INTERFACE ITcoObjectRestorer

(*~
	<docu>
		<summary>
			Ensures calling the <c>Restore()</c> method on the object entered.
			<para>
				<example>
				<note type="Example">
				<para>
					Possibility to use the fluent syntax.
				</para>
					<code>ChangeState(newState).RestoreObject(myFirstChildObject).RestoreObject(mySecondChildObject);</code>
				 </note>
				</example>
			</para>
		</summary>
	</docu>
~*)
METHOD RestoreObject : ITcoObjectRestorer
VAR_INPUT
	Obj : ITcoRestorable;
END_VAR
END_METHOD

END_INTERFACE

(* stored: Version 1.1.0.1
   Itf ITcoObjectRestorer: Id {0b3638df-96b7-05c9-2091-ef8947995aad}
   Method RestoreObject: Id {1cade283-565b-0b0e-0667-0d22a5ebb137} *)
